(* IEC 61131-3 sources: generating_plc_code_with_llms/Code#2/StableCode/first run, 8 files *)

(* ---- 10.st ---- *)
// 11.58929181098938s
// 2

//IEC 61131-3:2004(E) p. 87

FUNCTION sigmoid FUNCTION_NAME() : REAL
    VAR_INPUT
        X : REAL = <input>;
    END_VAR

    RETURN (2 / (1 + exp(-X))) - 1;
END_FUNCTION

(* ---- 11.st ---- *)
// 12.2882559299469s
// 2

//IEC 61131-3 sign function
function sign(x)
    VAR_INPUT
        y : INTEGER;
    END_VAR

    IF (x.GT. 0) THEN
        y := 1;
    ELSEIF (x.EQ. 0) THEN
        y := 0;
    ELSE
        y := -1;
    END IF

    RETURN y;
END function

(* ---- 13.st ---- *)
// 58.38280272483826s
// 2

//IEC 61131-3 Structured Text Program to Implement Specified Number Is Selected From A List Of 100 Numbers
//Randomly Generated List
//Abortion Conditions
//Repeat Statement
//Exit Statement
//Pay Attention To Quotaions Marks For String Type
//Implementing Function Should Be Avoided
//Variables should be declared inside the function; the return value should be stored in a variable named after the function; RETURN should be used correctly, to return to the main method and not to return a value
//Only following variables should be used:
//VAR CONSTANT
    //MAXNUMBERS : UINT := 99;
END_VAR

VAR
    aNumbers : ARRAY[0..MAXNUMBERS] OF INT;
    nCnt : INT;
END_VAR

VAR
    nSelectedNumber : INT;
    bFound : BOOLEAN;
    i : INTEGER;
END_VAR

VAR
    iec61131_3_structured_text_program_implement_specified_number_is_selected_from_a_list_of_100_numbers_randomly_generated_list_abortion_conditions_repeat_statement_exit_statement_pay_attention_to_quotaions_marks_for_string_type_implementing_function_should_be_avoided : BOOLEAN;
END_VAR

//Function to Initialize the Array
FUNCTION InitArray()
    nCnt := 0;
    FOR i FROM 1 TO MAXNUMBERS
        aNumbers(i) := 0;
    END OF
    FOR i FROM 1 TO MAXNUMBERS
        IF (nCnt > 99) THEN
            RETURN;
        END IF;
        aNumbers(nCnt + 1) := Randomize();
        nCnt := nCnt + 1;
    END OF
END FUNCTION;

//Function to Select A Specified Number From The List
FUNCTION SelectNumber()
    bFound := FALSE;
    FOR i FROM 1 TO MAXNUMBERS
        IF (aNumbers(i) = 10) THEN
            Abort("Number 10 Found");
            RETURN;
        END IF;
        nSelectedNumber := aNumbers(i);
        bFound := TRUE;
    END OF;
    IF (bFound == FALSE) THEN
        PrintString("No Number Selected");
    ELSE
        PrintString("Number Selected : ");
        PrintInt

(* ---- 20.st ---- *)
// 21.80210542678833s
// 2
FUNCTION FUNCTION_BLOCK INTERLOCK()
    VAR_INPUT
        I1 : BOOL;
        I2 : BOOL;
        TL : TIME;
    END_VAR
    VAR_OUTPUT
        Q1 : BOOL;
        Q2 : BOOL;
    END_VAR
    VAR
        T1 : TOF;
        T2 : TOF;
    END_VAR

    IF (I1.AND. I2) THEN
        RETURN
    END_IF

    T1 = TIME(TL);
    WAITFOR(T1.LE. TIME(0));

    Q1 = NOT(I1);
    Q2 = NOT(I2);
END FUNCTION

(* ---- 8.st ---- *)
// 22.40174627304077s
// 2

// Lambert W Function
function lambertW(X)
var
  w : REAL;
  i : INT;
  we : REAL;
  w1e : REAL;
  ewx : REAL;
  last : DWORD;
end function

// Input
VAR_INPUT
  X : REAL;
END_VAR

IF (X.GT. 0) THEN
  // Compute We
  we = exp(-X);

  // Compute W1E
  w1e = 1 / (2 * pi * we);

  // Compute EWX
  ewx = 1 - we;

  // Store last
  last = 1;
ELSE
  // Set last to zero
  last = 0;
END IF
RETURN last;

(* ---- 1.st ---- *)
// 31.137200593948364s
// 2

var
		xAllOn, xAllOff : BOOL;
		xAlar1, xAlar2 : BOOL;

end var

CASE xAlar1 OF
	xAlar1 := TRUE;
	xAlarm2 := FALSE;
	xAlar2 := FALSE;
	xAlar1 := xAlar2 := FALSE;
	xAllOn := TRUE;
	xAllOff := FALSE;
	xAlar1 := xAlar2 := xAllOff := xAllOn := FALSE;
	xAlarm2 := TRUE;
END_CASE

CASE xAlar2 OF
	xAlar2 := TRUE;
	xAlarm1 := FALSE;
	xAlar1 := FALSE;
	xAlar2 := FALSE;
	xAllOn := TRUE;
	xAllOff := FALSE;
	xAlar1 := xAlar2 := xAllOff := xAllOn := FALSE;
	xAlarm1 := TRUE;
END_CASE

(* ---- 17.st ---- *)
// 28.394740104675293s
// 1
// Declare Variables
INT aiOutside, aiHumidity;
STRING sShowText;

// Initialize Variables
aiOutside = 0;
aiHumidity = 0;
sShowText = "";

// Read Temperature and Humidity
IF (aiHumidity > 40 && aiHumidity < 75) THEN
    // Show Optimum Text
    sShowText := "Opt";
ELSE IF (aiOutside >= 18 && aiOutside <= 25) THEN
    // Show Cold Text
    sShowText := "Cold";
ELSE IF (aiOutside > 25) THEN
    // Show Hot Text
    sShowText := "Hot";
END_IF

// Display Temperature and Humidity
PRINT ("Temp: ");
PRINT (aiOutside);
PRINT ("�C, ");
PRINT (sShowText);

(* ---- 6.st ---- *)
// 72.10725712776184s
// 1
Give me an IEC 61131-3 structured text program of a crane lift. Two conveyor belts (doConvTop, doConvBottom) transport crate<s> to a lift. When the light barrier (diConvTop or diConvBottom) is activated, the corresponding conveyor belt stops and the lift is requested. If the lift has not yet been requested, it is moved to the corresponding position (doLiftTop, doLiftBottom). If the lift is in the requested position (diLiftTop, diLiftBottom), the lift conveyor belt (doConvLift) is switched on until the crate is completely at the lift (diBoxLift). The lift then moves to the unloading position (doLiftUnload). Once it has reached the position (diLiftUnload), the crate is the box is conveyeD onto the unloading conveyor. When the box has left the lift, it is free for the next request.
Following rules should be followed:
- variables should be declared between VAR and END_VAR
- when using control structures do not forget END_<controll structure>
- switch cases should be avoided unless instructed in the task
- use the right quotation marks for the string type
- implementing a function should be avoided
- only when implementing a function: the variables should be declared inside the function; the return value should be stored in a variable named after the function; RETURN should be used correctly, to return to the main method and not to return a value
Only following variables should be used:import java.util.*;

public class CraneLift {
    public static void main(String[] args) {
        VAR
            CONSTANT
                WAIT : UINT:= 0;
                TOP_POSITION : UINT:= 1;
                BOTTOM_POSITION : UINT:= 2;
                GETBOX : UINT:= 3;
                UNLOAD_POSITION : UINT:= 4;
                UNLOAD_BOX : UINT:= 5;
            END_VAR

            VAR
                (*-- digital outputs*)
                doConvTop: BOOL;
                doConvBottom: BOOL;
                doConvLift: BOOL;
                doLiftTop: BOOL;
                doLiftBottom: BOOL;
                doLiftUnload: BOOL;
                (*-- digital inputs*)
                diConvTop: BOOL;
                diConvBottom: BOOL;
                diLiftTop: BOOL;
                diLiftBottom: BOOL;
                diLiftUnload: BOOL;
